(* IEC 61131-3 sources: CodesysTest/alpha/export/FBs/Components/Motors/Applied Motion/FB_AppliedMotionStepServoEIPBaseQX.pou, 3 files *)

(* ---- Execute.m.st ---- *)
(*#-#-#-#-#-#-#-#-#-#---Declaration---#-#-#-#-#-#-#-#-#-#-#-#-#*)

METHOD Execute
VAR_INPUT
END_VAR
(*#-#-#-#-#-#-#-#-#-#---Implementation---#-#-#-#-#-#-#-#-#-#-#-#-#*)

//    Function Block: AppliedMotionStepServo
//    Description: This block provides an abstraction for a Ethernet I/P Applied Motion Step Servo
//    Created by: Ben Hess
//    Created Date: May 11th, 2018

// Use pointers for EIP memory register locations
driveInputs := ptrEIPInputs^;

ptrEIPOutputs^ := driveOutputs;
alarms(alarmCode := stepServoAlarmCodeRaw, faults := faults);

IF currentLimit = 0 THEN
	currentLimit := defaultCurrentSetpoint;
END_IF
//Map raw EIP Registers to parameters
absolutePositionSteps := driveInputs[6];
velocity := DINT_TO_INT(driveInputs[8]);
stepServoStatusRaw := DINT_TO_INT(driveInputs[0]);

driveOutputs[4] := velocitySetpoint;
driveOutputs[5] := pointToPointAccelSetpoint;
driveOutputs[6] := pointToPointDecelSetpoint;
driveOutputs[7] := distanceToMoveInSteps;
driveOutputs[8] := currentLimit;
driveOutputs[9] := sclCommand;
driveOutputs[10] := parameter1;
driveOutputs[11] := parameter2;
driveOutputs[12] := currentLimit;
driveOutputs[13] := currentLimit + 1;
driveOutputs[0] := commands.commandWord;
// Step servo command bits handler
commands();
//Convert Distance setpoint to steps.  Reverse polarity for display purposes if needed.

absolutePositonInches := (DINT_TO_REAL(absolutePositionSteps) / INT_TO_REAL(stepsPerInchSetpoint));

//Homing required from motor - for now just if there was an initialization seen.
homeRequiredIndication S= status.initializing OR Globals.firstScan OR _faulted OR driveInputs[11].0;

homingOSF(CLK := status.homing);
IF NOT driveInputs[11].0 THEN
	homeRequiredIndication := FALSE;
END_IF

commandSentONS(CLK := commands.commandSent);
IF commandSentONS.Q THEN
	commandSuccessful := TRUE;
END_IF

commandSuccessfulONS(CLK := commandSuccessful);
IF commandSuccessfulONS.Q THEN
	//parameter1 := 0;
	//velocitySetpoint := 0;
	//pointToPointAccelSetpoint := 0;
	//pointToPointDecelSetpoint := 0;
	//distanceToMoveInSteps := 0;
END_IF

IF _reset AND (status.driveFaulted OR status.alarmPresent) THEN
	commands.alarmReset := TRUE;
	_reset := FALSE;
END_IF

IF reversePolarity THEN
    absolutePositonInches := absolutePositonInches * -1;
END_IF

//Get Servo Status and unpack
status(statusCode := StepServoStatusRaw);

//Bit-packing for LONG types over Modbus

_faulted := status.driveFaulted OR status.alarmPresent OR commFail;

//Manual moves for motor
IF moveDistanceManualPB THEN
    MoveDistance(distance := distanceSetpointInches, acceleration := pointToPointAccelSetpoint, deceleration := pointToPointDecelSetpoint, velocity := velocitySetpoint);
    moveDistanceManualPB := FALSE;
END_IF

IF movePositionManualPB THEN
    MoveToPosition(position := distanceSetpointInches, acceleration := pointToPointAccelSetpoint, deceleration := pointToPointDecelSetpoint, velocity := velocitySetpoint);
    movePositionManualPB := FALSE;
END_IF

faults.commFail.faultTrigger := commFail AND Globals.machinePowerOK;
faults.notHomed.faultTrigger := homeRequiredIndication AND isHomable;

(* ---- ExecuteStoredProgram.m.st ---- *)
(*#-#-#-#-#-#-#-#-#-#---Declaration---#-#-#-#-#-#-#-#-#-#-#-#-#*)

METHOD ExecuteStoredProgram
VAR_INPUT
    (*Program number to execute*)
    programNumber    : INT;
END_VAR
(*#-#-#-#-#-#-#-#-#-#---Implementation---#-#-#-#-#-#-#-#-#-#-#-#-#*)

parameter1 := programNumber;
commands.SendQAndExecute := TRUE;

(* ---- MoveToPositionTorque.m.st ---- *)
(*#-#-#-#-#-#-#-#-#-#---Declaration---#-#-#-#-#-#-#-#-#-#-#-#-#*)

METHOD MoveToPositionTorque
VAR_INPUT
	(*Position to move to in inches*)
    position    : REAL;
    (*Acceleration in RPM/sec*)
    acceleration    : INT;
    (*Deceleration in RPM/sec*)
    deceleration    : INT;
    (*Velocity in .25RPM*)
    velocity    : INT;
	(*Current in .01A*)
	current : DINT;
END_VAR
(*#-#-#-#-#-#-#-#-#-#---Implementation---#-#-#-#-#-#-#-#-#-#-#-#-#*)

commandSuccessful := FALSE;

distanceToMoveInSteps := REAL_TO_DINT((position) * stepsPerInchSetpoint);
IF reversePolarity THEN
    distanceToMoveInSteps := distanceToMoveInSteps * -1;
END_IF

pointToPointAccelSetpoint := acceleration;
pointToPointDecelSetpoint := deceleration;
velocitySetpoint := velocity;
currentLimit := current;

commands.feedToPosition := TRUE;
THIS^.Execute();
